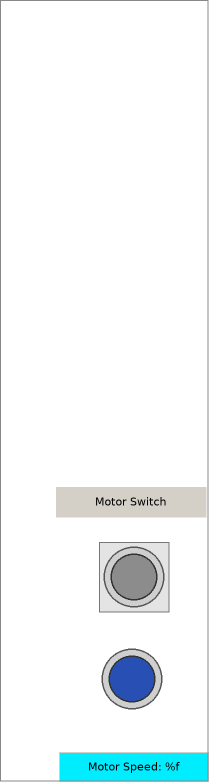
VISUALIZATION Visualization  // 209x782
    Lamp1 (97,644 70x70), variable: LenzeServoDrive.bButton, style: Lamp-Lamp1-Blue
    PushSwitch (99,542 70x70), variable: LenzeServoDrive.bButton, behaviour: TOGGLE, style: Switch-PushSwitch-Gray
    Textfield (56,487 150x30), "Motor Switch", colour toggle: LenzeServoDrive.bButton
    Textfield (59,752 150x30), "Motor Speed: %f", text variable: LenzeServoDrive.rActSpeed
END_VISUALIZATION

(* stored: Version 1.1.0.1, ProductVersion 3.1.4024.12
   Visu Visualization: Id {3bf92511-1793-4da0-811e-7e35aa2f7e4d} *)
